(* CODESYS project Property Example.project

Project tree, tasks and I/O mapping:
  Device : CODESYS SoftMotion RTE CX, 3S - Smart Software Solutions GmbH, order no. 309015, version 3.5.9.50
    application Application
      libraries: Standard, * (System)
      task MainTask (cyclic, interval 4 ms, priority 1) calls PLC_PRG
      program PLC_PRG [ST]
      function block FB1 [ST]: iTry, Set1
    SoftMotion General Axis Pool
*)

// Device/Application/PLC_PRG
PROGRAM PLC_PRG
VAR
	instance : FB1;
	instance2 :FB1;
	ivalue : INT;
	ivalue2 : int;
END_VAR

instance.iTry := 10;

ivalue := instance.iTry;

instance2.iTry := 5;

ivalue2 := instance2.iTry;

instance.iTry := instance2.iTry;

instance2.Set1(4);

END_PROGRAM

// Device/Application/FB1
FUNCTION_BLOCK FB1
VAR_INPUT
END_VAR
VAR_OUTPUT
END_VAR
VAR
	iVar : int := 0;
END_VAR

PROPERTY iTry : INT
SET
iVar := iTry;
END_SET
GET
iTry := iVar;
END_GET
END_PROPERTY

METHOD Set1
VAR_INPUT
	iInput :int;
END_VAR
THIS^.iVar := iInput;
END_METHOD

END_FUNCTION_BLOCK
